(* IEC 61131-3 sources: DirIOZip/, 2 files *)

(* ---- Types.typ ---- *)
TYPE
	DataObjectToFolder_typ : 	STRUCT
		ConvertToFile : DataObjToFile;
		Unzip : zipExtract;
		DeleteFile : FileDelete; (*Open a file and read its contents*)
		_Execute : BOOL;
		_DeleteTemp : BOOL;
		_Active : BOOL;
		_Finishing : BOOL;
		TempArchiveName : STRING[80];
	END_STRUCT;
	FolderToDataObject_typ : 	STRUCT
		Zip : zipArchive;
		ConvertToDataObject : FileToDataObj;
		DeleteFile : FileDelete; (*Open a file and read its contents*)
		_Execute : BOOL;
		_DeleteTemp : BOOL;
		_Active : BOOL;
		TempArchiveName : STRING[80];
	END_STRUCT;
END_TYPE

(* ---- DirIOZip.fun ---- *)
(********************************************************************
 * COPYRIGHT --
 ********************************************************************
 * Library: DirIOWrap
 * File: DirIOWrap.fun
 * Author: Josh
 * Created: April 24, 2015
 ********************************************************************
 * Functions and function blocks of library DirIOWrap
 ********************************************************************)

FUNCTION_BLOCK FolderToDataObj (* *) (*$GROUP=User,$CAT=User,$GROUPICON=User.png,$CATICON=User.png*)
	VAR_INPUT
		Execute : BOOL;
		FileDevice : STRING[80];
		TempFileDevice : STRING[80];
		FileName : STRING[80];
		DataObjectName : STRING[10];
	END_VAR
	VAR_OUTPUT
		Status : UINT;
	END_VAR
	VAR
		internal : FolderToDataObject_typ;
	END_VAR
END_FUNCTION_BLOCK

FUNCTION_BLOCK DataObjToFolder (*Convert a file to a dataobject*) (*$GROUP=User,$CAT=User,$GROUPICON=User.png,$CATICON=User.png*)
	VAR_INPUT
		Execute : BOOL;
		FileDevice : STRING[80];
		FileName : STRING[80];
		DataObjectName : STRING[10];
		DestPath : STRING[80];
		TempFileDevice : STRING[80];
	END_VAR
	VAR_OUTPUT
		Status : UINT;
	END_VAR
	VAR
		internal : DataObjectToFolder_typ;
	END_VAR
END_FUNCTION_BLOCK
